// TIA Portal V18 export
DATA_BLOCK "SS1_750A1_16DI_DI_Vars"   // DB11051
{ S7_Optimized_Access := 'FALSE' }
VERSION : 0.1
// stored: AutoNumber false, DBAccessibleFromOPCUA true, IsOnlyStoredInLoadMemory false, IsWriteProtectedInAS false
   VAR
      DI1 : "UDT_DIadv";   // Індикація живлення SS-1
      DI2 : "UDT_DIadv";   // HS Несправність системи опалення
      DI3 : "UDT_DIadv";   // HS Ін. 1- ст пальник К1
      DI4 : "UDT_DIadv";   // HS Ін. 2- ст пальник К1
      DI5 : "UDT_DIadv";   // Резерв
      DI6 : "UDT_DIadv";   // HS Аварія пальник К1
      DI7 : "UDT_DIadv";   // HS Ін. 1- ст пальник К2
      DI8 : "UDT_DIadv";   // HS Ін. 2- ст пальник К2
      DI9 { S7_SetPoint := 'True'} : "UDT_DIadv";   // HS Аварія пальник К2
      DI10 { S7_SetPoint := 'True'} : "UDT_DIadv";   // Резерв
      DI11 { S7_SetPoint := 'True'} : "UDT_DIadv";   // Резерв
      DI12 { S7_SetPoint := 'True'} : "UDT_DIadv";   // AHU NF Аварія ККБ
      DI13 { S7_SetPoint := 'True'} : "UDT_DIadv";   // AHU NF Ін. 1- ст. ККБ
      DI14 { S7_SetPoint := 'True'} : "UDT_DIadv";   // AHU NF Ін. 2- ст. ККБ
      DI15 { S7_SetPoint := 'True'} : "UDT_DIadv";   // Гот. роб. сист. обігр. дизельпроводу (10.211)
      DI16 { S7_SetPoint := 'True'} : "UDT_DIadv";   // AHU NF Гот. роб. обігр. пов. засл. (2.202)
   END_VAR
BEGIN
   DI3.cFuncSystemID := 10;
   DI3.cFuncVar := 25;
   DI4.cFuncSystemID := 10;
   DI4.cFuncVar := 26;
   DI5.cFuncSystemID := 10;
   DI5.cFuncVar := 27;
   DI6.cFuncSystemID := 100;
   DI6.cFuncVar := 11;
   DI7.cFuncSystemID := 100;
   DI7.cFuncVar := 12;
   DI8.cFuncSystemID := 10;
   DI8.cFuncVar := 24;
   DI9.cFuncSystemID := 10;
   DI9.cFuncVar := 22;
   DI10.xInversion := true;
   DI10.cFuncSystemID := 10;
   DI10.cFuncVar := 23;
   DI11.cFuncSystemID := 10;
   DI11.cFuncVar := 7;
   DI12.cFuncSystemID := 10;
   DI12.cFuncVar := 2;
   DI13.xInversion := true;
   DI13.cFuncSystemID := 10;
   DI13.cFuncVar := 3;
   DI14.cFuncSystemID := 10;
   DI14.cFuncVar := 5;
   DI15.xInversion := true;
   DI15.cFuncSystemID := 10;
   DI15.cFuncVar := 6;
END_DATA_BLOCK
